Fanuc KAREL source: CUST_READ_PARAMS.KL

PROGRAM CUST_READ_PARAMS
%STACKSIZE = 4000
%NOLOCKGROUP
%NOPAUSE=ERROR+COMMAND+TPENABLE
%ENVIRONMENT uif
%ENVIRONMENT sysdef
%ENVIRONMENT memo
%ENVIRONMENT kclop
%ENVIRONMENT bynam
%ENVIRONMENT fdev
%ENVIRONMENT flbt
%ENVIRONMENT regope
%INCLUDE klevccdf
%INCLUDE klevkeys
%INCLUDE klevkmsk
----POST ERRORS----
ROUTINE POSTERR(cause : STRING; status : INTEGER) &
FROM CUST_ERRORS
ROUTINE POST_CUST_ERR(cause : STRING) &
FROM CUST_ERRORS
----POST ERRORS----

----------------------------------------------
-----Read parameters with different types-----
-----INTEGER PARAMETERS-----
ROUTINE GET_TPE_INT_PARAMETER(number : INTEGER) : INTEGER
VAR
    data_type : INTEGER
    int_value : INTEGER
    real_value : REAL
    str_value : STRING[20]
    status : INTEGER
BEGIN
    GET_TPE_PRM(number, data_type, int_value, real_value, str_value, status)
    POSTERR('UNABLE TO READ PARAMETER', status)
    IF(data_type <> 1 ) THEN
        POST_CUST_ERR('PARAMETER SHOULD BE INTEGER ')
    ENDIF
    RETURN (int_value)
END GET_TPE_INT_PARAMETER
-----REAL PARAMETERS-----
ROUTINE GET_TPE_REAL_PARAMETER(number : INTEGER) : REAL
VAR
    data_type : INTEGER
    int_value : INTEGER
    real_value : REAL
    str_value : STRING[20]
    status : INTEGER
BEGIN
    GET_TPE_PRM(number, data_type, int_value, real_value, str_value, status)
    POSTERR('UNABLE TO READ PARAMETER', status)
    IF(data_type <> 2 ) THEN
        POST_CUST_ERR('PARAMETER SHOULD BE INTEGER ')
    ENDIF
    RETURN (real_value)
END GET_TPE_REAL_PARAMETER
-----STRING PARAMETERS-----
ROUTINE GET_TPE_STRING_PARAMETER(number : INTEGER) : STRING
VAR
    data_type : INTEGER
    int_value : INTEGER
    real_value : REAL
    str_value : STRING[20]
    status : INTEGER
BEGIN
    GET_TPE_PRM(number, data_type, int_value, real_value, str_value, status)
    POSTERR('UNABLE TO READ PARAMETER', status)
    IF(data_type <> 1 ) THEN
        POST_CUST_ERR('PARAMETER SHOULD BE INTEGER ')
    ENDIF
    RETURN (str_value)
END GET_TPE_STRING_PARAMETER
-----Read parameters with different types-----
----------------------------------------------
BEGIN
END CUST_READ_PARAMS
